// TwinCAT 3 PLC project shuttle_valve
// ProgramVersion: 3.1.4022.4
// libraries:
//   Tc2_EtherCAT, * (Beckhoff Automation GmbH)
//   Tc2_Standard, * (Beckhoff Automation GmbH)
//   Tc2_System, * (Beckhoff Automation GmbH)
//   Tc3_Module, * (Beckhoff Automation GmbH)
// project tree:
//   / PlcTask.TcTTO
//   POUs/ MAIN.TcPOU, POU.TcPOU
// real-time tasks:
//   TASK PlcTask: cycle T#10ms, priority 20, ADS port 350
// I/O:
//   DEVICE Device 1 (EtherCAT), AmsNetId 192.168.0.12.2.1
//     Box 1 (m1sa) [m1sa]
// variable links:
//   shuttle_valve/shuttle_valve Instance <-> Device 1 (EtherCAT)/Box 1 (m1sa)
//     PlcTask Inputs/MAIN.err_calibrated <-> Status process data mapping/err_calibrated
//     PlcTask Inputs/MAIN.err_dongle <-> Status process data mapping/err_dongle
//     PlcTask Inputs/MAIN.err_follow_error <-> Status process data mapping/err_follow_error
//     PlcTask Inputs/MAIN.err_force_minmax <-> Status process data mapping/err_force_minmax
//     PlcTask Inputs/MAIN.err_force_step <-> Status process data mapping/err_force_step
//     PlcTask Inputs/MAIN.err_masterhb <-> Status process data mapping/err_masterhb
//     PlcTask Inputs/MAIN.err_soc <-> Status process data mapping/err_soc
//     PlcTask Inputs/MAIN.sts_close_loop <-> Status process data mapping/close_loop
//     PlcTask Inputs/MAIN.sts_enable <-> Status process data mapping/enable
//     PlcTask Inputs/MAIN.sts_hb <-> Status process data mapping/slvhb
//     PlcTask Inputs/MAIN.sts_pwm1 <-> Status process data mapping/pwm1
//     PlcTask Inputs/MAIN.sts_pwm2 <-> Status process data mapping/pwm2
//     PlcTask Inputs/MAIN.sts_pwm3 <-> Status process data mapping/pwm3
//     PlcTask Inputs/MAIN.sts_rbX <-> Status process data mapping/force_rb_X
//     PlcTask Inputs/MAIN.sts_rbY <-> Status process data mapping/force_rb_Y
//     PlcTask Inputs/MAIN.sts_rbZ <-> Status process data mapping/force_rb_Z
//     PlcTask Inputs/MAIN.sts_spX <-> Status process data mapping/force_sp_X
//     PlcTask Inputs/MAIN.sts_spY <-> Status process data mapping/force_sp_Y
//     PlcTask Inputs/MAIN.sts_spZ <-> Status process data mapping/force_sp_Z
//     PlcTask Outputs/MAIN.cmd_close_loop <-> Control process data mapping/close_loop
//     PlcTask Outputs/MAIN.cmd_enable <-> Control process data mapping/enable
//     PlcTask Outputs/MAIN.cmd_hb <-> Control process data mapping/msthb
//     PlcTask Outputs/MAIN.cmd_spX <-> Control process data mapping/force_sp_X
//     PlcTask Outputs/MAIN.cmd_spY <-> Control process data mapping/force_sp_Y
//     PlcTask Outputs/MAIN.cmd_spZ <-> Control process data mapping/force_sp_Z

CONFIGURATION shuttle_valve
    RESOURCE PLC ON TwinCAT3
        TASK PlcTask(INTERVAL := T#10ms, PRIORITY := 20);
        PROGRAM MAIN WITH PlcTask : MAIN;
    END_RESOURCE
END_CONFIGURATION

// ---- POUs/MAIN.TcPOU
PROGRAM MAIN
VAR
	sts_spX AT %I*: REAL;
	sts_spY AT %I*: REAL;
	sts_spZ AT %I*: REAL;
	sts_rbX AT %I*: REAL;
	sts_rbY AT %I*: REAL;
	sts_rbZ AT %I*: REAL;
	sts_enable AT %I*: BOOL;
	sts_close_loop AT %I*: BOOL;
	sts_hb AT %I*: UDINT;
	sts_pwm1 AT %I*: REAL;
	sts_pwm2 AT %I*: REAL;
	sts_pwm3 AT %I*: REAL;
	
    err_force_minmax AT %I*: BOOL;
	err_force_step AT %I*: BOOL;
	err_follow_error AT %I*: BOOL;
	err_calibrated AT %I*: BOOL;
	err_masterhb AT %I*: BOOL;
	err_soc AT %I*: BOOL;
	err_dongle AT %I*: BOOL;
	
	cmd_spX AT %Q*: REAL;
	cmd_spY AT %Q*: REAL;
	cmd_spZ AT %Q*: REAL;
	cmd_enable AT %Q*: BOOL;
	cmd_close_loop AT %Q*: BOOL;
	cmd_hb AT %Q*: UDINT;
	
	cmd_clear_error : BOOL;
	pwm_flag : BOOL := TRUE;
END_VAR

MAIN.cmd_hb := MAIN.cmd_hb + 1;

IF pwm_flag = TRUE THEN
//	pwm_flag := FALSE;
	cmd_spX := 50;
	cmd_spY := 50;
	cmd_spZ := 50;	
END_IF

IF pwm_flag = FALSE THEN
//	pwm_flag := TRUE;
	cmd_spX := -50;
	cmd_spY := -50; 
	cmd_spZ := -50;	
END_IF

pwm_flag := NOT(pwm_flag);

END_PROGRAM

// ---- POUs/POU.TcPOU
PROGRAM POU
VAR
		

        fbSdoWrite      : FB_EcCoESdoWrite;
        //sNetId          : T_AmsNetId := ''; (* NetId of EtherCAT Master *) (* empty string == net id of the local device XXX does not work? *)
        sNetId          : T_AmsNetId := '192.168.2.15.2.1'; (* NetId of EtherCAT Master *)
        nSlaveAddr      : UINT := 1001; (* Port Number of EtherCAT Slave *)
        nIndex          : WORD := 16#8006; (* CoE Object Index *)
        nSubIndex       : BYTE := 1; (* Subindex of CoE Object *)
        bExecute        : BOOL; (* rising edge starts writing to the CoE Object *)
        bError          : BOOL;
        nErrId          : UDINT;
END_VAR


bExecute := MAIN.cmd_clear_error;

fbSdoWrite(
        sNetId          := sNetId,
        nSlaveAddr      := nSlaveAddr,
        nIndex          := nIndex,
        nSubIndex       := nSubIndex,
        pSrcBuf                 := ADR(MAIN.cmd_clear_error),
        cbBufLen                := SIZEOF(MAIN.cmd_clear_error),
        bExecute                := bExecute
);

IF NOT fbSdoWrite.bBusy THEN
        bExecute := FALSE;
        IF NOT bError THEN 
                (* write successful *)
                bError := FALSE;
                nErrId := 0;
        ELSE 
                (* write failed *)
                bError := fbSdoWrite.bError;
                nErrId := fbSdoWrite.nErrId;
        END_IF

        fbSdoWrite(bExecute := FALSE);
END_IF

END_PROGRAM
